SUBAPPLICATION SingleSelect (* Subapplication Type *)
  (* Standard: 61499-2 *)
  (* Version 1.1, 2026-09-27, Franz Höpfinger, Layout aufgeraeumt: AUI_DEMUX_4 in AUI_DEMUX umbenannt (der '_4' hatte keine Bedeutung), Baustein vertikal auf die Mitte der 5 ILOCK_T_FF_SR_AX-Kette zentriert, Event-Routing gleichmaessig aufgefaechert. *)
  (* Version 1.0, 2026-09-27, franz *)
  PACKAGE MyLib::sys;
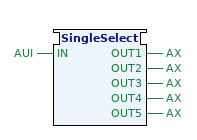
  SOCKETS
    IN : adapter::types::unidirectional::AUI;
  END_SOCKETS
  PLUGS
    OUT1 : adapter::types::unidirectional::AX;
    OUT2 : adapter::types::unidirectional::AX;
    OUT3 : adapter::types::unidirectional::AX;
    OUT4 : adapter::types::unidirectional::AX;
    OUT5 : adapter::types::unidirectional::AX;
  END_PLUGS
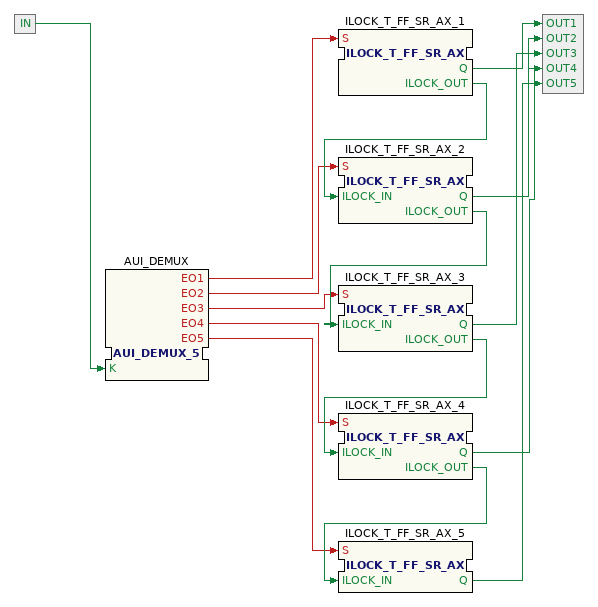
  FBS
    ILOCK_T_FF_SR_AX_1 : logiBUS::signalprocessing::interlock::ILOCK_T_FF_SR_AX;
    ILOCK_T_FF_SR_AX_2 : logiBUS::signalprocessing::interlock::ILOCK_T_FF_SR_AX;
    ILOCK_T_FF_SR_AX_3 : logiBUS::signalprocessing::interlock::ILOCK_T_FF_SR_AX;
    ILOCK_T_FF_SR_AX_4 : logiBUS::signalprocessing::interlock::ILOCK_T_FF_SR_AX;
    ILOCK_T_FF_SR_AX_5 : logiBUS::signalprocessing::interlock::ILOCK_T_FF_SR_AX;
    AUI_DEMUX : adapter::events::unidirectional::AUI_DEMUX_5;
  END_FBS
  EVENT_CONNECTIONS
    AUI_DEMUX.EO1 TO ILOCK_T_FF_SR_AX_1.S;
    AUI_DEMUX.EO2 TO ILOCK_T_FF_SR_AX_2.S;
    AUI_DEMUX.EO3 TO ILOCK_T_FF_SR_AX_3.S;
    AUI_DEMUX.EO4 TO ILOCK_T_FF_SR_AX_4.S;
    AUI_DEMUX.EO5 TO ILOCK_T_FF_SR_AX_5.S;
  END_CONNECTIONS
  ADAPTER_CONNECTIONS
    ILOCK_T_FF_SR_AX_1.Q TO OUT1;
    ILOCK_T_FF_SR_AX_2.Q TO OUT2;
    ILOCK_T_FF_SR_AX_3.Q TO OUT3;
    ILOCK_T_FF_SR_AX_4.Q TO OUT4;
    ILOCK_T_FF_SR_AX_5.Q TO OUT5;
    ILOCK_T_FF_SR_AX_1.ILOCK_OUT TO ILOCK_T_FF_SR_AX_2.ILOCK_IN;
    ILOCK_T_FF_SR_AX_2.ILOCK_OUT TO ILOCK_T_FF_SR_AX_3.ILOCK_IN;
    ILOCK_T_FF_SR_AX_3.ILOCK_OUT TO ILOCK_T_FF_SR_AX_4.ILOCK_IN;
    ILOCK_T_FF_SR_AX_4.ILOCK_OUT TO ILOCK_T_FF_SR_AX_5.ILOCK_IN;
    IN TO AUI_DEMUX.K;
  END_CONNECTIONS
END_SUBAPPLICATION
